Fanuc KAREL source: kb00052.KL

-- PROVISIONAL review KL for V770-1; original PC SHA256 520ba294efe4e8526b1a848d78b460331ebda19c5011741f4162c843bb449b07
-- Incomplete behavior may be omitted. Consult companion uncertainty JSON. Do not deploy.
PROGRAM KB00052
%NOLOCKGROUP
VAR
  P1 : INTEGER
  P2 : INTEGER
-- UNRESOLVED_DECL RESULT type=000106
BEGIN
  -- UNRESOLVED_PC offsets 5-12; opcodes 9D,23
  -- UNRESOLVED_PC offsets 17-24; opcodes 9D,23
  -- UNRESOLVED_PC offsets 29-58; opcodes 27,22,22,27,9D,76,7E,4A
  -- UNRESOLVED_PC offsets 63-67; opcodes 7F
END KB00052
